TYPE stManometerLabelSticking_TestData :
STRUCT
	bPressureCheckingEN: BOOL;		// Flaga włączająca sprawdzanie ciśnienia
	rSettingPressure:REAL;			// Wartość ciśniania do kalibracji
	rSettingPressureDeviation:REAL;	// Dopuszczalna odchyłka ciśnienia +/-	
END_STRUCT
END_TYPE

(* stored: Version 1.1.0.1, ProductVersion 3.1.4024.12
   DUT stManometerLabelSticking_TestData: Id {e3d5603f-1891-4d4c-a25c-6ad990ee48ea} *)
